FUNCTION_BLOCK Fb_UltrasonicSensor
VAR_INPUT
	i_UltraSonicAnalogInput		: INT;
	e_DistanceMode				: En_DistanceMode := En_DistanceMode.Default;
END_VAR
VAR_OUTPUT
	r_VoltageUltraSonicSensor	: REAL;
	i_AnalogOutput				: INT;
END_VAR
VAR
	l_UltraSonic				: DINT;
END_VAR
VAR CONSTANT
	MAX_VOLTAGE					: REAL := 10.0;
	MAX_INT						: INT := 32767;
END_VAR

// multiply by max voltage
l_UltraSonic := i_UltraSonicAnalogInput * REAL_TO_INT(MAX_VOLTAGE);

// divide by resolution
r_VoltageUltraSonicSensor := DINT_TO_REAL(l_UltraSonic) / INT_TO_REAL(MAX_INT);

// check distance mode and calculate
IF(e_DistanceMode = En_DistanceMode.NearerIsHigher) THEN
	l_UltraSonic := MAX_INT - i_UltraSonicAnalogInput;
ELSE
	l_UltraSonic := i_UltraSonicAnalogInput;
END_IF

// analog output, dint wont be larger than int at this point
i_AnalogOutput := DINT_TO_INT(l_UltraSonic);

END_FUNCTION_BLOCK

(* stored: Version 1.1.0.1, ProductVersion 3.1.4024.9
   POU Fb_UltrasonicSensor: Id {c18198f7-c06d-48df-ab56-66f4f3ccde48}, SpecialFunc None *)
